// TIA Portal V18 export
DATA_BLOCK "01_PushButton"   // DB3, F_DB
{ S7_Optimized_Access := 'TRUE'; DB_Accessible_From_OPC_UA := 'FALSE' }
// stored: DBAccessibleFromOPCUA false
   VAR
      AlwaysFALSE : Bool;   // Comment always false
      AlwaysTRUE : Bool := TRUE;
      "!!01_PushButton.SafetyBreaker1$$" : Bool;
      "!!01_PushButton.SafetyBreaker2$$" : Bool;
      "!!ITERATOR_STRINGS$$" : Bool;
   END_VAR
BEGIN
END_DATA_BLOCK
